TYPE ST_ComponentMyComponent_Config :
	STRUCT
	END_STRUCT
END_TYPE

(* stored: Version 1.1.0.1, ProductVersion 3.1.4024.12
   DUT ST_ComponentMyComponent_Config: Id {546ef656-d5c9-40c8-adca-7042f0e4cdc5} *)
